// TIA Portal V18 export
DATA_BLOCK "_ML3_importantPositionsRETAIN"   // DB67
{ S7_Optimized_Access := 'TRUE' }
VERSION : 0.1
// stored: AutoNumber true, DBAccessibleFromOPCUA true, IsOnlyStoredInLoadMemory false, IsRetainMemResEnabled false, IsWriteProtectedInAS false, MemoryReserve 100
   VAR RETAIN
      Load : "typePositions";
      Home : "typePositions";
      Control1 : "typePositions";
      Control2 : "typePositions";
   END_VAR
BEGIN
END_DATA_BLOCK
